PROGRAM progPITCntrl
VAR
	PIT_04_0100 : fbPIT;
END_VAR

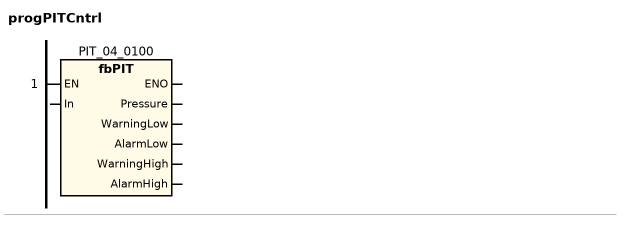
// NETWORK 1
PIT_04_0100(); // fbPIT

END_PROGRAM

(* stored: Version 1.1.0.1, ProductVersion 3.1.4022.17
   POU progPITCntrl: Id {7666ef51-fbb6-4fef-8cab-08398ca39c85}, SpecialFunc None *)
